# EPICS IOC start-up script: iocsh/AH401.iocsh
# ### AH401.iocsh ###

#- ###################################################
#- PREFIX         - IOC Prefix
#- INSTANCE       - Name of quadEM port instance to create
#- IP_ADDR        - IP address of AH401
#- QUADEM         - Location of quadEM module
#- ASYN           - Location of asyn module
#- MODEL          - Optional: AH401 Model (AH401B/AH401D)
#-                  Default: AH401B
#-
#- RING_SIZE      - Optional: Ring Size
#-                  Default: 10000
#-
#- QSIZE          - Optional: Queue size
#-                  Default: 20
#-
#- TSPOINTS       - Optional: Number of time series points
#-                  Default: 1000
#-
#- ###################################################

drvAsynIPPortConfigure("IP_$(INSTANCE)", "$(IP_ADDR)", 0, 0, 0)
asynOctetSetInputEos("IP_$(INSTANCE)",  0, "\r\n")
asynOctetSetOutputEos("IP_$(INSTANCE)", 0, "\r")

dbLoadRecords("$(ASYN)/db/asynRecord.db", "P=$(PREFIX), R=asyn_IP_$(INSTANCE),PORT=IP_$(INSTANCE),ADDR=0,OMAX=256,IMAX=256")

drvAHxxxConfigure("$(INSTANCE)", "IP_$(INSTANCE)", $(RING_SIZE=10000), "$(MODEL=AH401B)")

dbLoadRecords("$(QUADEM)/db/AH401B.template", "P=$(PREFIX), R=$(INSTANCE):, PORT=$(INSTANCE)")

iocshLoad("$(QUADEM)/iocsh/commonPlugins.iocsh")
